{attribute 'Tc2GvlVarNames'}
VAR_CONFIG
END_VAR

(* stored: Version 1.1.0.1, ProductVersion 3.1.4020.12
   GVL Variablen_Konfiguration: Id {2cccc8bd-14d8-4494-8e99-6934cd121992} *)
